// TwinCAT 3 PLC project PLC_code
// ProgramVersion: 3.1.4024.0
// CompilerDefines: VISU_USEWSTRING
// libraries:
//   Tc2_Math, * (Beckhoff Automation GmbH)
//   Tc2_MC2, * (Beckhoff Automation GmbH)
//   Tc2_NC, * (Beckhoff Automation GmbH)
//   Tc2_Standard, * (Beckhoff Automation GmbH)
//   Tc2_System, * (Beckhoff Automation GmbH)
//   Tc2_Utilities, * (Beckhoff Automation GmbH)
//   Tc3_Module, * (Beckhoff Automation GmbH)
// project tree:
//   / GlobalTextList.TcGTLO, PlcTask.TcTTO (not stored), Visualization Manager.TcVMO (not stored)
//   GVLs/ GVL.TcGVL, GVLLD.TcGVL (not stored)
//   POUs/ MAIN.TcPOU, ladder_logic_diagram.TcPOU, Meters_Travelled.TcPOU, SYSTEM.TcPOU, Safety_Zones.TcDUT
//   VISUs/ Charge_Velocity_Distance.TcVIS, Header.TcVIS, ImagePool.TcIPO (not stored), log_file.TcVIS (not stored), MainScreen.TcVIS, Nav.TcVIS (not stored), Nav_1.TcVIS (not stored), Safty_Zones_and_Modes.TcVIS
// real-time tasks:
//   TASK PlcTask: cycle T#10ms, priority 20, ADS port 350
//   TASK VISU_TASK: cycle T#200000us, priority 30, ADS port 351
// motion (NC):
//   TASK NC-Task 1 SAF: cycle T#2ms, priority 4, ADS port 501
//   TASK NC-Task 1 SVB: cycle T#10ms, priority 8, ADS port 511
//   AXIS Axis 1 (id 1)
//     Dynamic: Acceleration=5067.48, Deceleration=5067.48, Jerk=23830.8
//     Velo: RefSearch=14.56175, RefSync=14.56175, SlowManual=72.80875, FastManual=436.8525, Fast=1456.175, Maximum=1456.17
//     TargetPosControl: Range=20
//     OtherSettings: AllowMotionCmdToSlave=true, PulseDistancePos=20, PulseDistanceNeg=20
//     encoder EncType=19
//       EncPara: ScaleFactorNumerator=15.7, ScaleFactorDenominator=1048576, Inverse=true, MaxCount=#xffffffff
//     drive DrvType=16
//       DrvPara: Inverse=true, MaxCount=#xffffffff
//         Analog: VeloReferenz=1601.7925, VeloScale=32, TorqueSetpointScale=10, ScaleFactorActTorque=0.1
//         TimeComp: TaskDelayCycles=1
//     controller CtrType=1
//       CtrPara: PriorControlFactor=1
//         PosDiffControl: Range=40000
//         Observer: BandWidth=20
//   AXIS Axis 2 (id 2)
//     Dynamic: Acceleration=5067.48, Deceleration=5067.48, Jerk=23830.8
//     Velo: RefSearch=14.56175, RefSync=14.56175, SlowManual=72.80875, FastManual=436.8525, Fast=1456.175, Maximum=1456.17
//     TargetPosControl: Range=20
//     OtherSettings: AllowMotionCmdToSlave=true, PulseDistancePos=20, PulseDistanceNeg=20
//     encoder EncType=19
//       EncPara: ScaleFactorNumerator=15.7, ScaleFactorDenominator=1048576, MaxCount=#xffffffff
//     drive DrvType=16
//       DrvPara: MaxCount=#xffffffff
//         Analog: VeloReferenz=1601.7925, VeloScale=32, TorqueSetpointScale=10, ScaleFactorActTorque=0.1
//         TimeComp: TaskDelayCycles=1
//     controller CtrType=1
//       CtrPara: PriorControlFactor=1
//         PosDiffControl: Range=40000
//         Observer: BandWidth=20
//   AXIS Axis 3 (id 3)
//     Dynamic: Acceleration=14588.3136, Deceleration=14588.3136, Jerk=43764.9408
//     Velo: RefSearch=97.255424, RefSync=97.255424, SlowManual=486.27712, FastManual=2917.66272, Fast=9725.5424, Maximum=9725.5424
//     OtherSettings: AllowMotionCmdToSlave=true
//     encoder EncType=19
//       EncPara: ScaleFactorNumerator=104.8576, ScaleFactorDenominator=1048576, MaxCount=#xffffffff
//     drive DrvType=16
//       DrvPara: MaxCount=#xffffffff
//         Analog: VeloReferenz=10698.09664, VeloScale=32, TorqueSetpointScale=10, ScaleFactorActTorque=0.1
//         TimeComp: TaskDelayCycles=1
//     controller CtrType=1
//       CtrPara: PriorControlFactor=1
//         PosDiffControl: Range=10
//         Observer: BandWidth=20
// variable links:
//   PLC_code/PLC_code Instance <-> NC-Task 1 SAF/Axes/Axis 1
//     PlcTask Inputs/MAIN.AxisB.NcToPlc <-> Outputs/ToPlc
//     PlcTask Outputs/MAIN.AxisB.PlcToNc <-> Inputs/FromPlc
//   PLC_code/PLC_code Instance <-> NC-Task 1 SAF/Axes/Axis 2
//     PlcTask Inputs/MAIN.AxisA.NcToPlc <-> Outputs/ToPlc
//     PlcTask Outputs/MAIN.AxisA.PlcToNc <-> Inputs/FromPlc

// ---- POUs/Safety_Zones.TcDUT
TYPE Safety_Zones :
STRUCT
	Front_back_white_zone : BOOL := FALSE ;
	Front_back_red_zone : BOOL := FALSE ;
	Front_back_purple_zone : BOOL := TRUE ;
	Front_back_grey_pink_zone : BOOL := TRUE ;
	
END_STRUCT
END_TYPE

// ---- GVLs/GVL.TcGVL
{attribute 'qualified_only'}
VAR_GLOBAL
	
	GetLocalSystemTime : FB_LocalSystemTime;
	SystemDateTime : STRING;
	SystemDate : STRING;
	SystemTime : STRING;
	SystemMinutes : STRING;
	SystemSeconds : STRING ; 
END_VAR

// ---- POUs/MAIN.TcPOU
PROGRAM MAIN
VAR
	// ntp.beckhoff-cloud.com
	// time.windows.com
	Lidar_zones:  Safety_Zones; 
	encoderPosition AT  %I* : UDINT;
	actualAxisPosition AT  %I* : LREAL;
	actualAxisPositionA AT  %I* : LREAL;
	Left_Encoder : LREAL;
	Right_Encoder : LREAL;
	setPositionA AT  %I* : LREAL ;
	setPositionB AT  %I* : LREAL ;
	AxisB : AXIS_REF;
	AxisA : AXIS_REF;
	timer : TON;
	SetTimeToRtcTime : Nt_SetTimeToRtcTime  ;
	// Motor 1
	McPower : MC_Power;
	McReset : MC_Reset;
	McJogging : MC_Jog;
	McVelocity : MC_MoveVelocity;
	McStop :  MC_Stop;
	McHalt : MC_Halt;
	McSetPositionA: MC_SetPosition;
	McSetPosition: MC_SetPosition;
	McPosition : MC_ReadActualPosition;
	McPositionA : MC_ReadActualPosition;
	

	// Motor 2
	McPowerA : MC_Power;
	McResetA : MC_Reset;
	McJoggingA : MC_Jog;
	McVelocityA : MC_MoveVelocity;
	McStopA :  MC_Stop;
	McHaltA : MC_Halt;
	
	CppVelocityValue : DINT;
	CppVelocityCmd : DINT;
	RightVelocityValue : REAL;
	LeftVelocityValue : REAL;
	RightVelocityCmd : REAL;
	LeftVelocityCmd : REAL;
	RightVelocity_meters : REAL;
	LeftVelocity_meters : REAL;
	acc : REAL:=0;
	dcc : REAL:=0;
	jk	: REAL:=0;
	myvelocity : DINT;
	cppvar AT %I* : BOOL;
	pypositive AT %I* : BOOL;
	pynegative AT %I* : BOOL;
	pyturnright AT %I* : BOOL;
	pyturnleft AT %I* : BOOL;
	state : DINT;
	stop AT %I* : BOOL;
	fright AT %I* : BOOL;
	bright AT %I* : BOOL;
	fleft AT %I* : BOOL;
	bleft AT %I* : BOOL;

	ChargeSignal       AT %Q* : BOOL;
	Lift_UP            AT %Q* : BOOL:= FALSE;
	Lift_DOWN          AT %Q* : BOOL;
	Lift_UP_Signal	   AT %M* : BOOL;
	Lift_DOWN_Signal   AT %M* : BOOL;
	Lift_Stop          AT %M* : BOOL;
	FrontLidarWarning  AT %I* : BOOL;
	BackLidarWarning   AT %I* : BOOL;

	stopvalue : BOOL;
	Acceleration: LREAL;
	Options: INT;
	nVAR: REAL;
	
	//Lidar Zones
	zon_1_set          AT %M* : BOOL; 
	zon_2_set          AT %M* : BOOL; 
	zon_3_set          AT %M* : BOOL; 
	zon_4_set          AT %M* : BOOL; 
	zon_5_set          AT %M* : BOOL; 
	zon_6_set          AT %M* : BOOL;    
	
	PLC_Minutes : INT;
	PLC_Seconds : INT;
	velocity_seconds : INT;
	velocity_minutes : INT;
	time_difference : INT := 0 ;
	abs_time_difference : INT := 0 ;
	velocity_timeout : BOOL := FALSE ;
	
	NETID  : T_AmsNetId := '192.168.0.176.1.1' ;
    SET    : BOOL;
    TMOUT  : TIME := DEFAULT_ADS_TIMEOUT;
	
	first_pc_time_reading: INT;
	second_pc_time_reading: INT;
END_VAR

SYSTEM();
Meters_Travelled();
Ladder_Logic_Diagram();

SetTimeToRtcTime( NETID := '192.168.0.176.1.1' ,
					SET := TRUE,
					TMOUT:= DEFAULT_ADS_TIMEOUT);


//PLC_Minutes := STRING_TO_INT (GVL.SystemMinutes);
//PLC_Seconds := STRING_TO_INT (GVL.SystemSeconds);
//time_difference := PLC_Seconds  - velocity_seconds  ;
//abs_time_difference := ABS(time_difference);
IF GVLLD.first_time_read THEN
first_pc_time_reading := STRING_TO_INT (GVL.SystemSeconds);	
END_IF
IF GVLLD.second_time_read THEN
second_pc_time_reading := STRING_TO_INT (GVL.SystemSeconds);
END_IF
// Axis B Left Motor
AxisB.ReadStatus();
McPower(Axis:=AxisB,Enable := TRUE,Enable_Positive := TRUE, Enable_Negative := TRUE);
McSetPosition(Axis:= AxisB,Execute:= TRUE, Position := setPositionA);
McPosition(Axis := AxisB,Enable := TRUE );
actualAxisPosition := McPosition.Position;
Left_Encoder := actualAxisPosition ;

// Axis A Right Motor
AxisA.ReadStatus();
McPowerA(Axis:=AxisA,Enable := TRUE,Enable_Positive := TRUE, Enable_Negative := TRUE);
McSetPositionA(Axis:= AxisA,Execute:= TRUE, Position := setPositionB);
McPositionA(Axis := AxisA,Enable := TRUE );
actualAxisPositionA := McPositionA.Position;
Right_Encoder := actualAxisPositionA ;

CppVelocityCmd := CppVelocityValue;
RightVelocity_meters := RightVelocityCmd /1000 ;
LeftVelocity_meters := LeftVelocityCmd / 1000 ;
IF NOT GVLLD.view_safety THEN
	RightVelocityCmd := 0;
	LeftVelocityCmd := 0;
	ELSE IF NOT FrontLidarWarning OR NOT BackLidarWarning THEN
		RightVelocityCmd := RightVelocityValue * 0.9;
		LeftVelocityCmd := LeftVelocityValue * 0.9;
	ELSE IF FrontLidarWarning OR BackLidarWarning THEN
		RightVelocityCmd := RightVelocityValue;
		LeftVelocityCmd := LeftVelocityValue;
		END_IF
	END_IF
END_IF

stopvalue := stop;



CASE state OF 
	0: 	
		state := 10;
	10: 
		McReset(Axis := AxisB,Execute := FALSE);
		McResetA(Axis := AxisA,Execute := FALSE);
		McReset(Axis := AxisB,Execute := TRUE);
		McResetA(Axis := AxisA,Execute := TRUE);
		IF McReset.Done AND McResetA.Done  THEN
			state := 20;
		ELSIF NOT McReset.Done OR NOT McResetA.Done THEN 
			McReset(Axis := AxisB,Execute := FALSE);
			McResetA(Axis := AxisA,Execute := FALSE);
			McReset(Axis := AxisB,Execute := TRUE);
			McResetA(Axis := AxisA,Execute := TRUE);
			state := 20;
		END_IF
		
	20: 
	
		McPowerA(Axis:=AxisA,Enable := TRUE,Enable_Positive := TRUE, Enable_Negative := TRUE);
		McPower(Axis:=AxisB,Enable := TRUE,Enable_Positive := TRUE, Enable_Negative := TRUE);
		IF McPower.Status AND McPowerA.Status THEN
			state :=50;
		END_IF
		
	
	//CPP Function Block
//	40: 
		
//		McVelocityA (Axis:= AxisA,
//					Execute := cppvar,
//					Velocity := CppVelocityCmd,
//						Acceleration := acc,
//						Deceleration := dcc,
//						Jerk := jk,
//					Direction := MC_Direction.MC_Positive_Direction ) ;
//		McVelocity (Axis:= AxisB,
//					Execute := cppvar,
//					Velocity := CppVelocityCmd,
//						Acceleration := acc,
//						Deceleration := dcc,
//						Jerk := jk,
//					Direction := MC_Direction.MC_Positive_Direction ) ;
//		McVelocityA (Axis:= AxisA,
//					Execute := cppvar,
//					Velocity := CppVelocityCmd,
//						Acceleration := acc,
//						Deceleration := dcc,
//						Jerk := jk,
//					Direction := MC_Direction.MC_Negative_Direction ) ;
//		McVelocity (Axis:= AxisB,
//					Execute := cppvar,
//					Velocity := CppVelocityCmd,
//						Acceleration := acc,
//						Deceleration := dcc,
//						Jerk := jk,
//					Direction := MC_Direction.MC_Negative_Direction ) ;
//		IF stopvalue THEN
//			McVelocity(Axis := AxisB, Execute := FALSE); 
//			McVelocityA(Axis := AxisA, Execute := FALSE); 
//			state := 900;
//		END_IF
//		IF fright OR fleft OR bright OR bleft THEN 
//			McVelocity(Axis := AxisB, Execute := FALSE);
//			McVelocityA(Axis := AxisA, Execute := FALSE);
//			state := 50;
//		END_IF
		
		
	//Python Function Block
	50: 
		// POSİTİVE
		IF AxisA.Status.Error OR AxisB.Status.Error THEN 
			McReset(Axis := AxisB,Execute := FALSE);
			McResetA(Axis := AxisA,Execute := FALSE);
			McReset(Axis := AxisB,Execute := TRUE);
			McResetA(Axis := AxisA,Execute := TRUE);
//			state :=0;
		END_IF
		IF stopvalue THEN
			
			McVelocity(Axis := AxisB, Execute := FALSE); 
			McVelocityA(Axis := AxisA, Execute := FALSE);
			state := 900;
		END_IF
		IF GVLLD.auto_charge_signal THEN   
   			McVelocity(Axis := AxisB, Execute := FALSE);    
			McVelocityA(Axis := AxisA, Execute := FALSE);
  			state := 400;  
		END_IF

		
//		IF time_difference >  2 AND abs_time_difference < 57 THEN
		IF first_pc_time_reading = second_pc_time_reading THEN
			velocity_timeout := TRUE;
			LeftVelocityValue := 0 ;
			RightVelocityValue := 0 ;
			RightVelocityCmd := RightVelocityValue;
			LeftVelocityCmd := LeftVelocityValue;
			McVelocityA (Axis:= AxisA,
						Execute := FALSE,
						Velocity := RightVelocityCmd,
						Acceleration := acc,
						Deceleration := dcc,
						Jerk := jk,
						Direction := MC_Direction.MC_Positive_Direction ) ;
			McVelocityA (Axis:= AxisA,
						Execute := TRUE,
						Velocity := RightVelocityCmd,
						Acceleration := acc,
						Deceleration := dcc,
						Jerk := jk,
						Direction := MC_Direction.MC_Negative_Direction ) ;
			McVelocity (Axis:= AxisB,
						Execute := FALSE,
						Velocity := LeftVelocityCmd,
						Acceleration := acc,
						Deceleration := dcc,
						Jerk := jk,
						Direction := MC_Direction.MC_Positive_Direction ) ;
			McVelocity (Axis:= AxisB,
						Execute := TRUE,
						Velocity := LeftVelocityCmd,
						Acceleration := acc,
						Deceleration := dcc,
						Jerk := jk,
						Direction := MC_Direction.MC_Negative_Direction ) ;
		state :=50;
		ELSE
		velocity_timeout := FALSE;

		IF RightVelocityCmd >= 0 THEN
			fright := TRUE;
			bright := FALSE;
		END_IF
		IF RightVelocityCmd < 0 THEN
			fright := FALSE;
			bright := TRUE;
		END_IF
		IF LeftVelocityCmd >= 0 THEN 
			fleft := TRUE;
			bleft := FALSE;
		END_IF
		IF LeftVelocityCmd < 0 THEN
			fleft := FALSE;
			bleft := TRUE;
		END_IF

		McVelocity (Axis:= AxisB,
						Execute := bleft,
						Velocity := ABS(LeftVelocityCmd),
						Acceleration := acc,
						Deceleration := dcc,
						Jerk := jk,
						Direction := MC_Direction.MC_Negative_Direction ) ;
		McVelocity (Axis:= AxisB,
						Execute := fleft,
						Velocity := ABS(LeftVelocityCmd),
						Acceleration := acc,
						Deceleration := dcc,
						Jerk := jk,
						Direction := MC_Direction.MC_Positive_Direction ) ;
		McVelocityA (Axis:= AxisA,
						Execute := bright,
						Velocity := ABS(RightVelocityCmd),
						Acceleration := acc,
						Deceleration := dcc,
						Jerk := jk,
						Direction := MC_Direction.MC_Negative_Direction ) ;
		McVelocityA (Axis:= AxisA,
						Execute := fright, 
						Velocity := ABS(RightVelocityCmd),
						Acceleration := acc,
						Deceleration := dcc,
						Jerk := jk,
						Direction := MC_Direction.MC_Positive_Direction ) ;
	state :=50;
		END_IF
		
			

		
		IF cppvar THEN 
			McVelocity(Axis := AxisB, Execute := FALSE);
			McVelocityA(Axis := AxisA, Execute := FALSE);
			state := 40;
		END_IF
	400:  
		IF AxisA.Status.Error OR AxisB.Status.Error THEN 
		   	McReset(Axis := AxisB,Execute := FALSE);   
			McResetA(Axis := AxisA,Execute := FALSE);
		   	McReset(Axis := AxisB,Execute := TRUE);   
			McResetA(Axis := AxisA,Execute := TRUE);
  		END_IF
    	McStop(Axis := AxisB, Execute := TRUE);
  		McStopA(Axis := AxisA, Execute := TRUE);  
  		IF NOT GVLLD.auto_charge_signal THEN   
			McStop(Axis := AxisB, Execute := FALSE); 
			McVelocity(Axis := AxisB, Execute := FALSE);    
			McStopA(Axis := AxisA, Execute := FALSE); 
			McVelocityA(Axis := AxisA, Execute := FALSE);    
			state := 50;
  		END_IF
	900:
		IF AxisA.Status.Error OR AxisB.Status.Error THEN 
			McReset(Axis := AxisB,Execute := FALSE);
			McResetA(Axis := AxisA,Execute := FALSE);
			McReset(Axis := AxisB,Execute := TRUE);
			McResetA(Axis := AxisA,Execute := TRUE);
		END_IF
		McStop(Axis := AxisB, Execute := TRUE);
		McStopA(Axis := AxisA, Execute := TRUE);
		IF fright OR fleft OR bright OR bleft OR pyturnleft OR cppvar THEN
			McStop(Axis := AxisB, Execute := FALSE); 
			McVelocity(Axis := AxisB, Execute := FALSE); 
			McStopA(Axis := AxisA, Execute := FALSE); 
			McVelocityA(Axis := AxisA, Execute := FALSE); 
			state := 50;
		END_IF
		
		
		
END_CASE

END_PROGRAM

// ---- POUs/SYSTEM.TcPOU
PROGRAM SYSTEM
VAR
END_VAR

GVL.GetLocalSystemTime(
	sNetID := ,
	bEnable := TRUE,
	dwCycle := 1,
	dwOpt:= ,
	tTimeout:= ,
	bValid =>,
	systemTime=>,
	tzID=>);
	
GVL.SystemDateTime := SYSTEMTIME_TO_STRING(GVL.GetLocalSystemTime.systemTime);
GVL.SystemDate := MID(STR:= GVL.SystemDateTime,LEN:=10,POS:=1);
GVL.SystemTime := MID(STR:= GVL.SystemDateTime,LEN:=8,POS:=12);
GVL.SystemMinutes := MID(STR:= GVL.SystemDateTime,LEN:=2,POS:=15);
GVL.SystemSeconds := MID(STR:= GVL.SystemDateTime,LEN:=2,POS:=18);

END_PROGRAM

// ---- POUs/Meters_Travelled.TcPOU
PROGRAM Meters_Travelled
VAR
	
	// Right Encoder 
	r_read_first_encoder : BOOL := TRUE;
	r_first_read : LREAL ;
	r_second_read : LREAL ;
	r_diff_read : LREAL ;
	r_prev_diff_read : LREAL := 0 ; 
	r_total_diff_read : LREAL ;
	r_meters_travelled : LREAL ;
	r_encoder_ticks : LREAL := 0  ;
//////////////////////////////////////////////////
	//Left Encoder 
	l_read_first_encoder : BOOL := TRUE;
	l_first_read : LREAL ;
	l_second_read : LREAL ;
	l_diff_read : LREAL ;
	l_prev_diff_read : LREAL := 0 ; 
	l_total_diff_read : LREAL ;
	l_meters_travelled : LREAL ;
	l_encoder_ticks : LREAL := 0  ;


END_VAR

r_encoder_ticks :=  MAIN.Right_Encoder ;
IF r_read_first_encoder THEN 
	r_first_read := r_encoder_ticks ;
END_IF
r_second_read := r_encoder_ticks ;
r_diff_read := ABS (r_second_read - r_first_read) ; 
IF r_diff_read < 0.001 THEN
	r_diff_read := 0 ;
END_IF
r_total_diff_read := r_diff_read + r_prev_diff_read ;
r_meters_travelled := r_total_diff_read / 1000  ;
r_prev_diff_read := r_total_diff_read ;
r_first_read := r_second_read ;
r_read_first_encoder := FALSE ;

l_encoder_ticks :=  MAIN.Left_Encoder;
IF l_read_first_encoder THEN 
	l_first_read := l_encoder_ticks ;
END_IF
l_second_read := l_encoder_ticks ;
l_diff_read := ABS (l_second_read - l_first_read) ;
IF l_diff_read < 0.001 THEN
	l_diff_read := 0 ;
END_IF 
l_total_diff_read := l_diff_read + l_prev_diff_read ;
l_meters_travelled := l_total_diff_read / 1000  ;
l_prev_diff_read := l_total_diff_read ;
l_first_read := l_second_read ;
l_read_first_encoder := FALSE ;

END_PROGRAM

// ---- POUs/ladder_logic_diagram.TcPOU
PROGRAM ladder_logic_diagram 
VAR
	t2s: TIME := TIME#3S;
	t0s: TIME := TIME#0S;
	Timer: TON;
	input : BOOL;
	output : BOOL; 
	TON_Reset: TON;
	TON_set: TON;
	TON_0: TON;
	TON_Trig: TON;
	TON_Autonomous: TON;
	TON_Manual: TON;
	TON_Lock: TON;
	Robot_Mode_Timer: TON;
	liftUP: TON;
	liftDOWN: TON;
	load_button  AT %I* : BOOL ;
	load_active AT %Q*: BOOL;
	trigger AT %M* : BOOL ;
	T: TIME;
	TON_1: TON;
	TON2: TON;
	TON_3: TON;
	activate_time_read: BOOL;
	TON_4: TON;
	second_read_triggered: BOOL;
	first_read_triggered: BOOL;
	TON_5: TON;
	TON_6: TON;
	TON_7: TON;
END_VAR
VAR // added by the converter: edge detectors and wires of the graphical bodies
    _rt1 : R_TRIG;
    _w1 : BOOL;
END_VAR

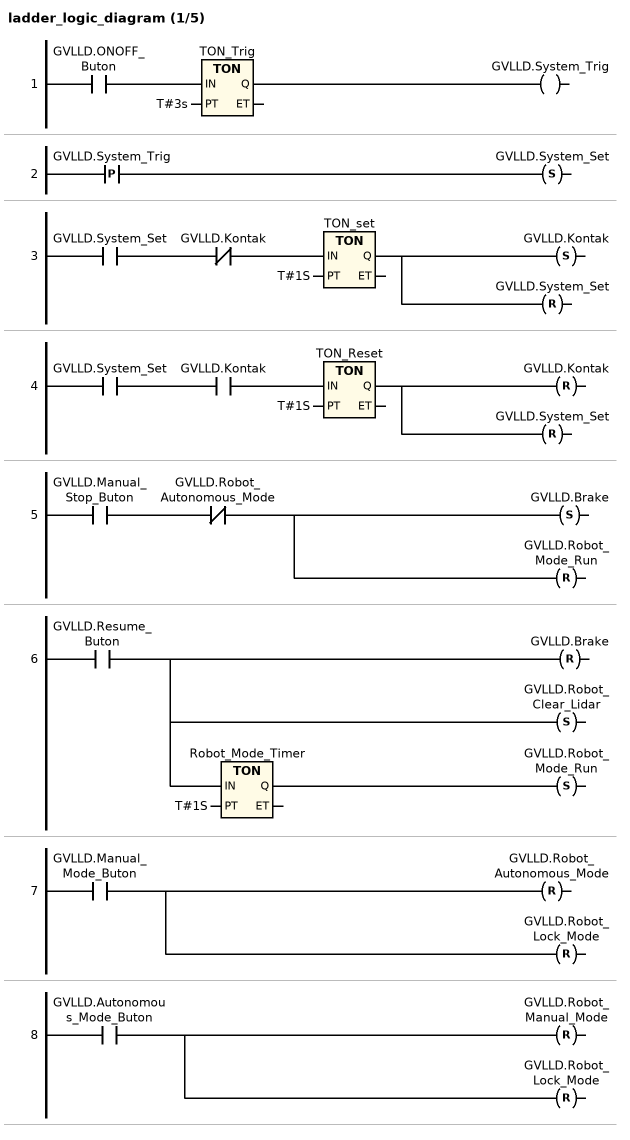
// NETWORK 1
TON_Trig(IN := GVLLD.ONOFF_Buton, PT := T#3s); // TON
GVLLD.System_Trig := TON_Trig.Q;

// NETWORK 2
_rt1(CLK := GVLLD.System_Trig);
GVLLD.System_Set S= _rt1.Q;

// NETWORK 3
TON_set(IN := GVLLD.System_Set AND NOT GVLLD.Kontak, PT := T#1S); // TON
GVLLD.Kontak S= TON_set.Q;
GVLLD.System_Set R= TON_set.Q;

// NETWORK 4
TON_Reset(IN := GVLLD.System_Set AND GVLLD.Kontak, PT := T#1S); // TON
GVLLD.Kontak R= TON_Reset.Q;
GVLLD.System_Set R= TON_Reset.Q;

// NETWORK 5
_w1 := GVLLD.Manual_Stop_Buton AND NOT GVLLD.Robot_Autonomous_Mode;
GVLLD.Brake S= _w1;
GVLLD.Robot_Mode_Run R= _w1;

// NETWORK 6
GVLLD.Brake R= GVLLD.Resume_Buton;
GVLLD.Robot_Clear_Lidar S= GVLLD.Resume_Buton;
Robot_Mode_Timer(IN := GVLLD.Resume_Buton, PT := T#1S); // TON
GVLLD.Robot_Mode_Run S= Robot_Mode_Timer.Q;

// NETWORK 7
GVLLD.Robot_Autonomous_Mode R= GVLLD.Manual_Mode_Buton;
GVLLD.Robot_Lock_Mode R= GVLLD.Manual_Mode_Buton;

// NETWORK 8
GVLLD.Robot_Manual_Mode R= GVLLD.Autonomous_Mode_Buton;
GVLLD.Robot_Lock_Mode R= GVLLD.Autonomous_Mode_Buton;

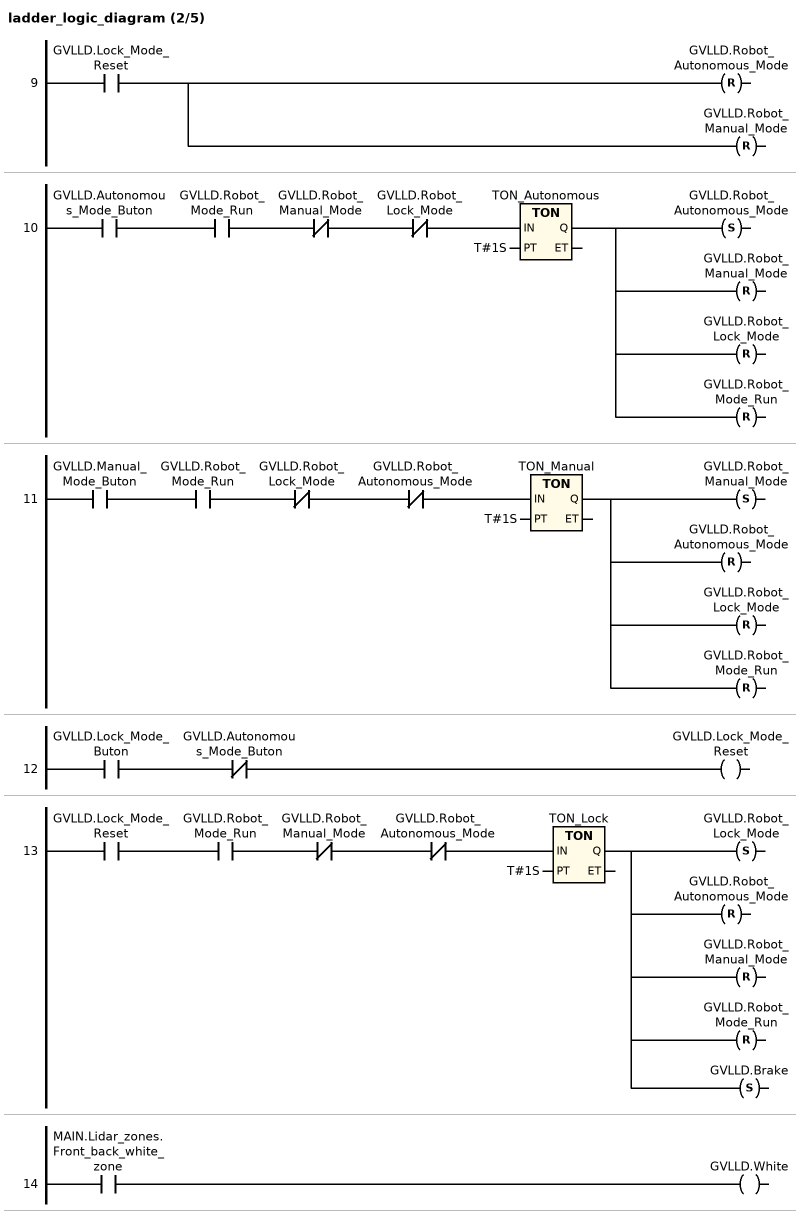
// NETWORK 9
GVLLD.Robot_Autonomous_Mode R= GVLLD.Lock_Mode_Reset;
GVLLD.Robot_Manual_Mode R= GVLLD.Lock_Mode_Reset;

// NETWORK 10
TON_Autonomous(IN := GVLLD.Autonomous_Mode_Buton AND GVLLD.Robot_Mode_Run AND NOT GVLLD.Robot_Manual_Mode AND NOT GVLLD.Robot_Lock_Mode, PT := T#1S); // TON
GVLLD.Robot_Autonomous_Mode S= TON_Autonomous.Q;
GVLLD.Robot_Manual_Mode R= TON_Autonomous.Q;
GVLLD.Robot_Lock_Mode R= TON_Autonomous.Q;
GVLLD.Robot_Mode_Run R= TON_Autonomous.Q;

// NETWORK 11
TON_Manual(IN := GVLLD.Manual_Mode_Buton AND GVLLD.Robot_Mode_Run AND NOT GVLLD.Robot_Lock_Mode AND NOT GVLLD.Robot_Autonomous_Mode, PT := T#1S); // TON
GVLLD.Robot_Manual_Mode S= TON_Manual.Q;
GVLLD.Robot_Autonomous_Mode R= TON_Manual.Q;
GVLLD.Robot_Lock_Mode R= TON_Manual.Q;
GVLLD.Robot_Mode_Run R= TON_Manual.Q;

// NETWORK 12
GVLLD.Lock_Mode_Reset := GVLLD.Lock_Mode_Buton AND NOT GVLLD.Autonomous_Mode_Buton;

// NETWORK 13
TON_Lock(IN := GVLLD.Lock_Mode_Reset AND GVLLD.Robot_Mode_Run AND NOT GVLLD.Robot_Manual_Mode AND NOT GVLLD.Robot_Autonomous_Mode, PT := T#1S); // TON
GVLLD.Robot_Lock_Mode S= TON_Lock.Q;
GVLLD.Robot_Autonomous_Mode R= TON_Lock.Q;
GVLLD.Robot_Manual_Mode R= TON_Lock.Q;
GVLLD.Robot_Mode_Run R= TON_Lock.Q;
GVLLD.Brake S= TON_Lock.Q;

// NETWORK 14
GVLLD.White := MAIN.Lidar_zones.Front_back_white_zone;

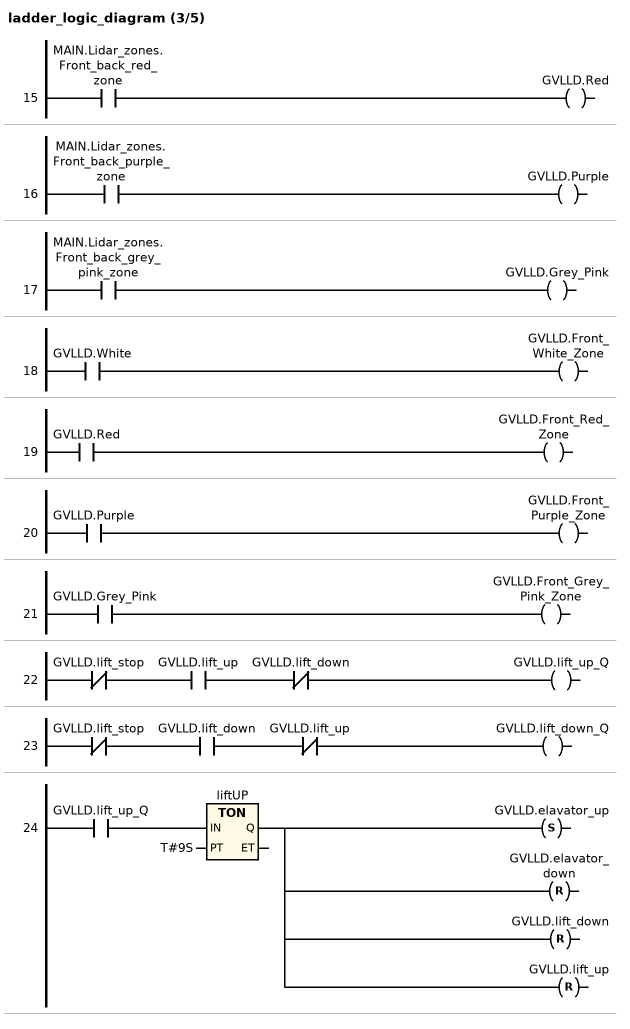
// NETWORK 15
GVLLD.Red := MAIN.Lidar_zones.Front_back_red_zone;

// NETWORK 16
GVLLD.Purple := MAIN.Lidar_zones.Front_back_purple_zone;

// NETWORK 17
GVLLD.Grey_Pink := MAIN.Lidar_zones.Front_back_grey_pink_zone;

// NETWORK 18
GVLLD.Front_White_Zone := GVLLD.White;

// NETWORK 19
GVLLD.Front_Red_Zone := GVLLD.Red;

// NETWORK 20
GVLLD.Front_Purple_Zone := GVLLD.Purple;

// NETWORK 21
GVLLD.Front_Grey_Pink_Zone := GVLLD.Grey_Pink;

// NETWORK 22
GVLLD.lift_up_Q := NOT GVLLD.lift_stop AND GVLLD.lift_up AND NOT GVLLD.lift_down;

// NETWORK 23
GVLLD.lift_down_Q := NOT GVLLD.lift_stop AND GVLLD.lift_down AND NOT GVLLD.lift_up;

// NETWORK 24
liftUP(IN := GVLLD.lift_up_Q, PT := T#9S); // TON
GVLLD.elavator_up S= liftUP.Q;
GVLLD.elavator_down R= liftUP.Q;
GVLLD.lift_down R= liftUP.Q;
GVLLD.lift_up R= liftUP.Q;

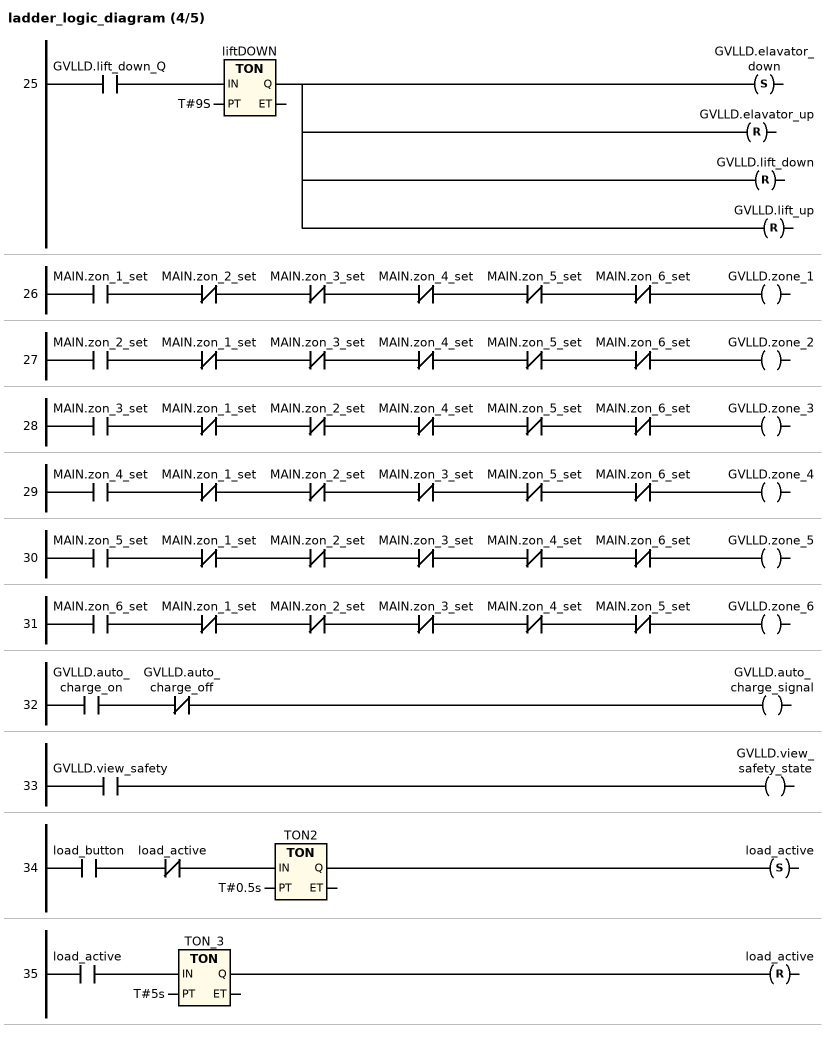
// NETWORK 25
liftDOWN(IN := GVLLD.lift_down_Q, PT := T#9S); // TON
GVLLD.elavator_down S= liftDOWN.Q;
GVLLD.elavator_up R= liftDOWN.Q;
GVLLD.lift_down R= liftDOWN.Q;
GVLLD.lift_up R= liftDOWN.Q;

// NETWORK 26
GVLLD.zone_1 := MAIN.zon_1_set AND NOT MAIN.zon_2_set AND NOT MAIN.zon_3_set AND NOT MAIN.zon_4_set AND NOT MAIN.zon_5_set AND NOT MAIN.zon_6_set;

// NETWORK 27
GVLLD.zone_2 := MAIN.zon_2_set AND NOT MAIN.zon_1_set AND NOT MAIN.zon_3_set AND NOT MAIN.zon_4_set AND NOT MAIN.zon_5_set AND NOT MAIN.zon_6_set;

// NETWORK 28
GVLLD.zone_3 := MAIN.zon_3_set AND NOT MAIN.zon_1_set AND NOT MAIN.zon_2_set AND NOT MAIN.zon_4_set AND NOT MAIN.zon_5_set AND NOT MAIN.zon_6_set;

// NETWORK 29
GVLLD.zone_4 := MAIN.zon_4_set AND NOT MAIN.zon_1_set AND NOT MAIN.zon_2_set AND NOT MAIN.zon_3_set AND NOT MAIN.zon_5_set AND NOT MAIN.zon_6_set;

// NETWORK 30
GVLLD.zone_5 := MAIN.zon_5_set AND NOT MAIN.zon_1_set AND NOT MAIN.zon_2_set AND NOT MAIN.zon_3_set AND NOT MAIN.zon_4_set AND NOT MAIN.zon_6_set;

// NETWORK 31
GVLLD.zone_6 := MAIN.zon_6_set AND NOT MAIN.zon_1_set AND NOT MAIN.zon_2_set AND NOT MAIN.zon_3_set AND NOT MAIN.zon_4_set AND NOT MAIN.zon_5_set;

// NETWORK 32
GVLLD.auto_charge_signal := GVLLD.auto_charge_on AND NOT GVLLD.auto_charge_off;

// NETWORK 33
GVLLD.view_safety_state := GVLLD.view_safety;

// NETWORK 34
TON2(IN := load_button AND NOT load_active, PT := T#0.5s); // TON
load_active S= TON2.Q;

// NETWORK 35
TON_3(IN := load_active, PT := T#5s); // TON
load_active R= TON_3.Q;

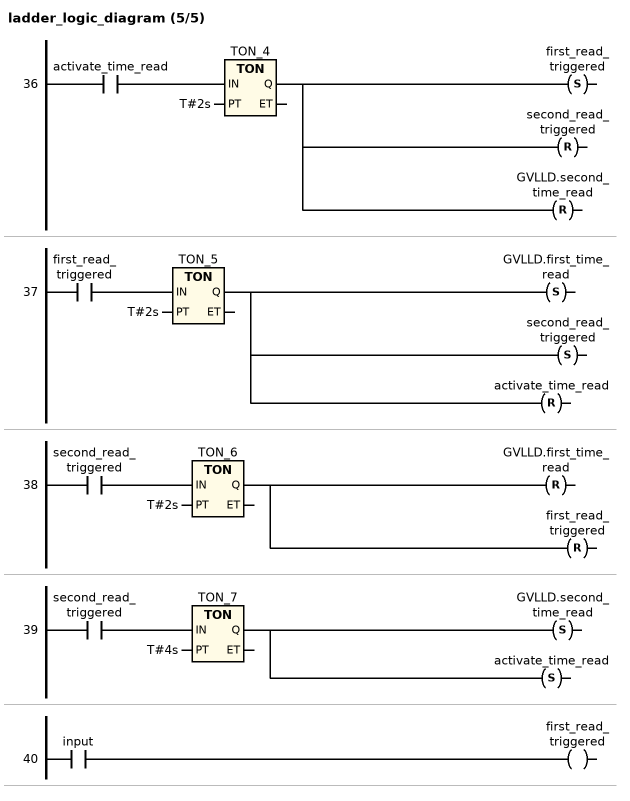
// NETWORK 36
TON_4(IN := activate_time_read, PT := T#2s); // TON
first_read_triggered S= TON_4.Q;
second_read_triggered R= TON_4.Q;
GVLLD.second_time_read R= TON_4.Q;

// NETWORK 37
TON_5(IN := first_read_triggered, PT := T#2s); // TON
GVLLD.first_time_read S= TON_5.Q;
second_read_triggered S= TON_5.Q;
activate_time_read R= TON_5.Q;

// NETWORK 38
TON_6(IN := second_read_triggered, PT := T#2s); // TON
GVLLD.first_time_read R= TON_6.Q;
first_read_triggered R= TON_6.Q;

// NETWORK 39
TON_7(IN := second_read_triggered, PT := T#4s); // TON
GVLLD.second_time_read S= TON_7.Q;
activate_time_read S= TON_7.Q;

// NETWORK 40
first_read_triggered := input;

END_PROGRAM

// ---- GlobalTextList.TcGTLO
TEXTLIST GlobalTextList
  644 = ' SCREEN 2'
  104 = ' To Main Screen'
  960 = ' TO SCREEN 1'
  399 = '%s'
  895 = 'Autonomous Mode '
  782 = 'Charge Status'
  893 = 'EPIC ROBOTICS'
  305 = 'EPİK ROBOTİK'
  788 = 'FALSE'
  362 = 'ISMAIL'
  853 = 'Left Motor Speed'
  796 = 'LIAMSI'
  856 = 'Lidar Zones'
  21 = 'Lock Mode '
  813 = 'Log File'
  133 = 'LİDAR ZONES'
  986 = 'm'
  529 = 'm/s'
  702 = 'MAIN'
  295 = 'MAIN SCREEN'
  175 = 'Main Screen'
  479 = 'Manual Mode '
  585 = 'Meters Travelled Left Motor'
  636 = 'Meters Travelled Right Motor'
  371 = 'Right Motor Speed'
  740 = 'Robot Modes'
  762 = 'Safety Zones '
  498 = 'SCREEN 1'
  469 = 'SCREEN 2'
  695 = 'TO MAIN'
  904 = 'TO SCREEN 2'
  821 = 'To Screen 2 '
  669 = 'To Screen1'
  897 = 'Velocity & Charge'
  387 = 'Zone 1'
  65 = 'Zone 2'
  171 = 'Zone 3'
  249 = 'Zone 4'
  28 = 'Zone 5'
  296 = 'Zone 6'
  142 = 'ZONES'
  201 = 'Zones & Modes'
END_TEXTLIST

// ---- VISUs/Charge_Velocity_Distance.TcVIS
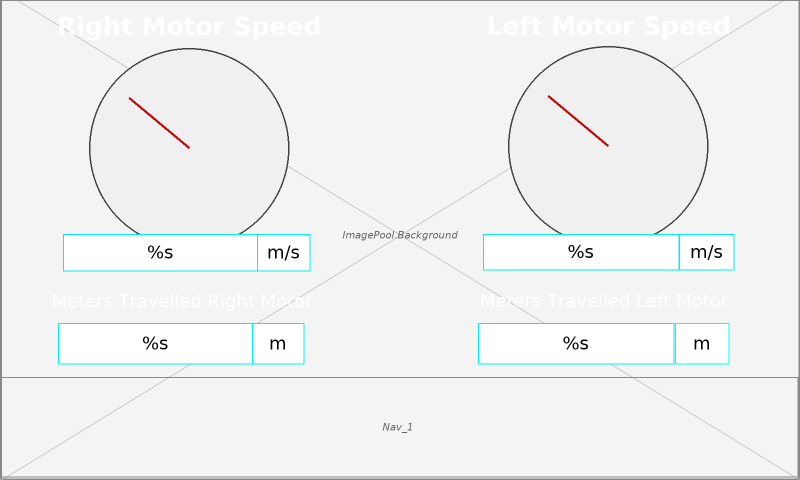
VISUALIZATION Charge_Velocity_Distance  // 800x480
    Image (1,-10 799x490), image: ImagePool.Background
    Meter180 (14,48 350x200), value: MAIN.RightVelocityValue, style: Meter-Meter180-Green, scale format: %.1f, scale 0..0.7
        p518627256: m/s
    Meter180 (433,46 350x200), value: MAIN.LeftVelocityValue, style: Meter-Meter180-Green, scale format: %.1f, scale 0..0.7
        p518627256: m/s
    RoundedRectangle (57,10 265x32), "Right Motor Speed"
    RoundedRectangle (478,10 262x31), "Left Motor Speed"
    Textfield (63,234 195x37), "%s", text variable: MAIN.RightVelocityValue
    Textfield (483,234 196x36), "%s", text variable: MAIN.LeftVelocityValue
    Rectangle (257,234 53x37), "m/s"
    BarDisplayImage (823,379 336x111), style: BarDisplayImage-Yellow, scale format: %.1f, scale 0..100
    RoundedRectangle (463,281 282x40), "Meters Travelled Left Motor"
    Textfield (58,323 195x41), "%s", text variable: Meters_Travelled.r_meters_travelled
    Rectangle (252,323 52x41), "m"
    RoundedRectangle (41,282 282x39), "Meters Travelled Right Motor"
    Textfield (478,323 196x41), "%s", text variable: Meters_Travelled.l_meters_travelled
    Rectangle (675,323 54x41), "m"
    Rectangle (679,234 55x36), "m/s"
    Frame (-2,377 800x100)
        shows Nav_1()
END_VISUALIZATION

// ---- VISUs/Header.TcVIS
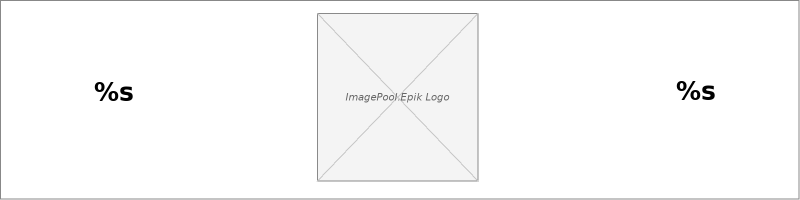
VISUALIZATION Header  // 800x200
    Image (317,13 161x168), image: ImagePool.Epik Logo
    Textfield (601,41 190x99), "%s", text variable: GVL.SystemTime
    Textfield (8,43 212x97), "%s", text variable: GVL.SystemDate
END_VISUALIZATION

// ---- VISUs/MainScreen.TcVIS
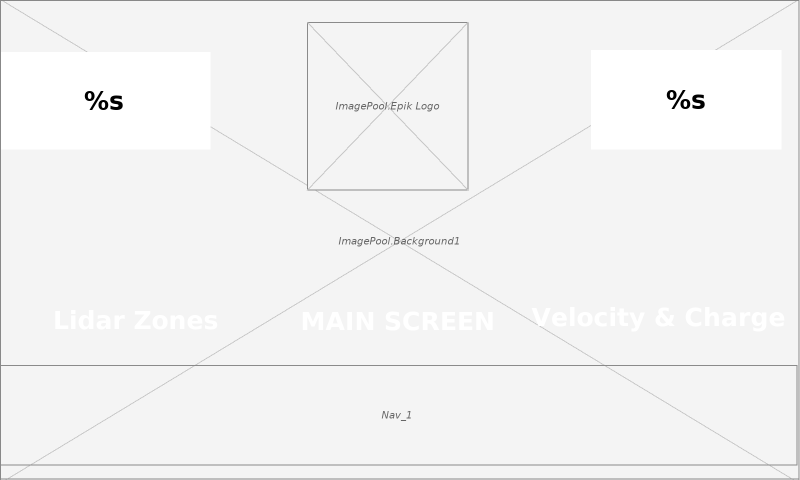
VISUALIZATION MainScreen  // 800x480
    Image (0,-1 799x484), image: ImagePool.Background1
    Frame (-10,9 800x200)
        shows Header()
    Frame (-3,365 800x100)
        shows Nav_1()
    RoundedRectangle (291,289 214x64), "MAIN SCREEN"
    RoundedRectangle (531,285 255x64), "Velocity & Charge"
    RoundedRectangle (29,288 214x64), "Lidar Zones"
END_VISUALIZATION

// ---- VISUs/Safty_Zones_and_Modes.TcVIS
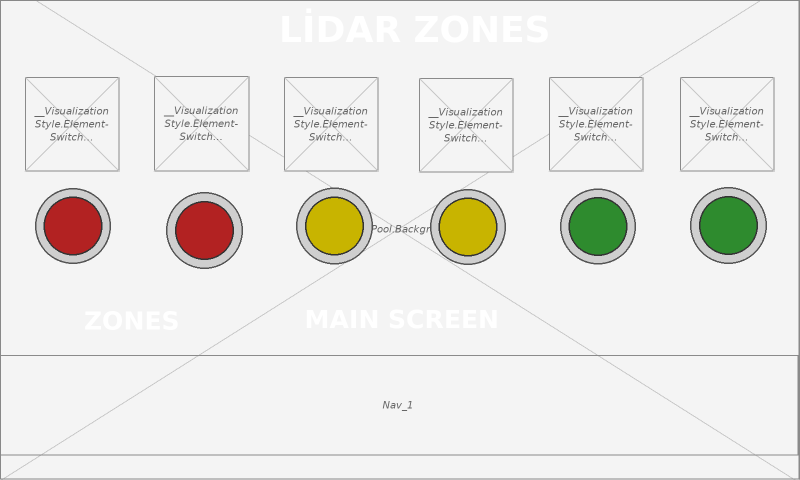
VISUALIZATION Safty_Zones_and_Modes  // 800x480
    Image (-4,-25 804x508), image: ImagePool.Background
    Lamp1 (29,182 88x88), variable: GVLLD.zone_1, invisible if: FALSE, style: Lamp-Lamp1-Red
    Lamp1 (160,182 89x97), variable: GVLLD.zone_2, invisible if: FALSE, style: Lamp-Lamp1-Red
    Lamp1 (290,181 89x90), variable: GVLLD.zone_3, invisible if: FALSE, style: Lamp-Lamp1-Yellow
    Lamp1 (424,182 88x90), variable: GVLLD.zone_4, invisible if: FALSE, style: Lamp-Lamp1-Yellow
    Lamp1 (554,182 88x89), variable: GVLLD.zone_5, invisible if: FALSE, style: Lamp-Lamp1-Green
    Lamp1 (684,181 89x89), tooltip "FALSE", variable: GVLLD.zone_6, style: Lamp-Lamp1-Green
    RoundedRectangle (154,8 522x43), "LİDAR ZONES"
    Frame (-2,355 800x100)
        shows Nav_1()
    Image (680,77 94x94), invisible if: FALSE, input disabled if: FALSE
        OnMouseClick: execute {
            MAIN.Lidar_zones.Front_back_white_zone:= TRUE;
            MAIN.Lidar_zones.Front_back_red_zone:= TRUE;
            MAIN.Lidar_zones.Front_back_purple_zone:= FALSE;
            MAIN.Lidar_zones.Front_back_grey_pink_zone:= FALSE;
            MAIN.zon_1_set:= FALSE;
            MAIN.zon_2_set:= FALSE;
            MAIN.zon_3_set:= FALSE;
            MAIN.zon_4_set:= FALSE;
            MAIN.zon_5_set:= FALSE;
            MAIN.zon_6_set:= TRUE;
        }
    Image (549,77 94x94), invisible if: FALSE, input disabled if: FALSE
        OnMouseClick: execute {
            MAIN.Lidar_zones.Front_back_white_zone:= TRUE;
            MAIN.Lidar_zones.Front_back_red_zone:= FALSE;
            MAIN.Lidar_zones.Front_back_purple_zone:= TRUE;
            MAIN.Lidar_zones.Front_back_grey_pink_zone:= FALSE;
            MAIN.zon_1_set:= FALSE;
            MAIN.zon_2_set:= FALSE;
            MAIN.zon_3_set:= FALSE;
            MAIN.zon_4_set:= FALSE;
            MAIN.zon_5_set:= TRUE;
            MAIN.zon_6_set:= FALSE;
        }
    Image (419,78 94x94), invisible if: FALSE, input disabled if: FALSE
        OnMouseClick: execute {
            MAIN.Lidar_zones.Front_back_white_zone:= FALSE;
            MAIN.Lidar_zones.Front_back_red_zone:= TRUE;
            MAIN.Lidar_zones.Front_back_purple_zone:= TRUE;
            MAIN.Lidar_zones.Front_back_grey_pink_zone:= FALSE;
            MAIN.zon_1_set:= FALSE;
            MAIN.zon_2_set:= FALSE;
            MAIN.zon_3_set:= FALSE;
            MAIN.zon_4_set:= TRUE;
            MAIN.zon_5_set:= FALSE;
            MAIN.zon_6_set:= FALSE;
        }
    Image (284,77 94x94), invisible if: FALSE, input disabled if: FALSE
        OnMouseClick: execute {
            MAIN.Lidar_zones.Front_back_white_zone:= TRUE;
            MAIN.Lidar_zones.Front_back_red_zone:= FALSE;
            MAIN.Lidar_zones.Front_back_purple_zone:= FALSE;
            MAIN.Lidar_zones.Front_back_grey_pink_zone:= TRUE;
            MAIN.zon_1_set:= FALSE;
            MAIN.zon_2_set:= FALSE;
            MAIN.zon_3_set:= TRUE;
            MAIN.zon_4_set:= FALSE;
            MAIN.zon_5_set:= FALSE;
            MAIN.zon_6_set:= FALSE;
        }
    Image (154,76 95x95), invisible if: FALSE, input disabled if: FALSE
        OnMouseClick: execute {
            MAIN.Lidar_zones.Front_back_white_zone:= FALSE;
            MAIN.Lidar_zones.Front_back_red_zone:= TRUE;
            MAIN.Lidar_zones.Front_back_purple_zone:= FALSE;
            MAIN.Lidar_zones.Front_back_grey_pink_zone:= TRUE;
            MAIN.zon_1_set:= FALSE;
            MAIN.zon_2_set:= TRUE;
            MAIN.zon_3_set:= FALSE;
            MAIN.zon_4_set:= FALSE;
            MAIN.zon_5_set:= FALSE;
            MAIN.zon_6_set:= FALSE;
        }
    Image (25,77 94x94), invisible if: FALSE, input disabled if: FALSE
        OnMouseClick: execute {
            MAIN.Lidar_zones.Front_back_white_zone:= FALSE;
            MAIN.Lidar_zones.Front_back_red_zone:= FALSE;
            MAIN.Lidar_zones.Front_back_purple_zone:= TRUE;
            MAIN.Lidar_zones.Front_back_grey_pink_zone:= TRUE;
            MAIN.zon_1_set:= TRUE;
            MAIN.zon_2_set:= FALSE;
            MAIN.zon_3_set:= FALSE;
            MAIN.zon_4_set:= FALSE;
            MAIN.zon_5_set:= FALSE;
            MAIN.zon_6_set:= FALSE;
        }
        OnMouseDown: execute {  }
    RoundedRectangle (286,298 232x42), "MAIN SCREEN"
    RoundedRectangle (15,300 234x41), "ZONES"
END_VISUALIZATION
